KUKA KRL program: di_seitlichFUENFZEHN_unkomp.src, di_seitlichFUENFZEHN_unkomp.dat

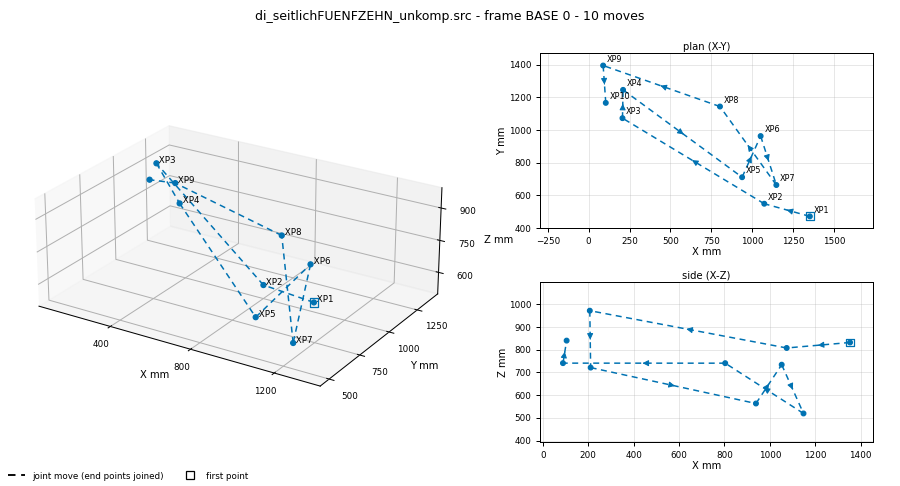
[picture p0: tool path of di_seitlichFUENFZEHN_unkomp.src in frame BASE 0, 10 of 12 moves have a stored position in this frame; points joined in program order, loops and branches not executed]
--- di_seitlichFUENFZEHN_unkomp.src ---
&ACCESS RV
&REL 1
&PARAM EDITMASK = *
&PARAM TEMPLATE = C:\KRC\Roboter\Template\vorgabe
DEF di_s_FZ_unkomp( )
;FOLD INI;%{PE}
  ;FOLD BASISTECH INI
    GLOBAL INTERRUPT DECL 3 WHEN $STOPMESS==TRUE DO IR_STOPM ( )
    INTERRUPT ON 3
    BAS (#INITMOV,0 )
  ;ENDFOLD (BASISTECH INI)
  ;FOLD USER INI
    ;Make your modifications here

  ;ENDFOLD (USER INI)
;ENDFOLD (INI)

;FOLD PTP HOME Vel=10 % DEFAULT;%{PE}%R 8.3.40,%MKUKATPBASIS,%CMOVE,%VPTP,%P 1:PTP, 2:HOME, 3:, 5:10, 7:DEFAULT
$BWDSTART=FALSE
PDAT_ACT=PDEFAULT
FDAT_ACT=FHOME
BAS(#PTP_PARAMS,10)
$H_POS=XHOME
PTP XHOME
;ENDFOLD

WAIT FOR IS_KEY_PRESSED(12)

;FOLD PTP P1 Vel=30 % PDAT1 Tool[11]:jan_ba Base[0];%{PE}%R 8.3.40,%MKUKATPBASIS,%CMOVE,%VPTP,%P 1:PTP, 2:P1, 3:, 5:30, 7:PDAT1
$BWDSTART=FALSE
PDAT_ACT=PPDAT1
FDAT_ACT=FP1
BAS(#PTP_PARAMS,30)
PTP XP1
;ENDFOLD

WAIT FOR IS_KEY_PRESSED(12)

;FOLD PTP P2 Vel=30 % PDAT2 Tool[11]:jan_ba Base[0];%{PE}%R 8.3.40,%MKUKATPBASIS,%CMOVE,%VPTP,%P 1:PTP, 2:P2, 3:, 5:30, 7:PDAT2
$BWDSTART=FALSE
PDAT_ACT=PPDAT2
FDAT_ACT=FP2
BAS(#PTP_PARAMS,30)
PTP XP2
;ENDFOLD

WAIT FOR IS_KEY_PRESSED(12)

;FOLD PTP P3 Vel=30 % PDAT3 Tool[11]:jan_ba Base[0];%{PE}%R 8.3.40,%MKUKATPBASIS,%CMOVE,%VPTP,%P 1:PTP, 2:P3, 3:, 5:30, 7:PDAT3
$BWDSTART=FALSE
PDAT_ACT=PPDAT3
FDAT_ACT=FP3
BAS(#PTP_PARAMS,30)
PTP XP3
;ENDFOLD

WAIT FOR IS_KEY_PRESSED(12)

;FOLD PTP P4 Vel=30 % PDAT4 Tool[11]:jan_ba Base[0];%{PE}%R 8.3.40,%MKUKATPBASIS,%CMOVE,%VPTP,%P 1:PTP, 2:P4, 3:, 5:30, 7:PDAT4
$BWDSTART=FALSE
PDAT_ACT=PPDAT4
FDAT_ACT=FP4
BAS(#PTP_PARAMS,30)
PTP XP4
;ENDFOLD

WAIT FOR IS_KEY_PRESSED(12)

;FOLD PTP P5 Vel=30 % PDAT5 Tool[11]:jan_ba Base[0];%{PE}%R 8.3.40,%MKUKATPBASIS,%CMOVE,%VPTP,%P 1:PTP, 2:P5, 3:, 5:30, 7:PDAT5
$BWDSTART=FALSE
PDAT_ACT=PPDAT5
FDAT_ACT=FP5
BAS(#PTP_PARAMS,30)
PTP XP5
;ENDFOLD

WAIT FOR IS_KEY_PRESSED(12)


;FOLD PTP P6 Vel=30 % PDAT6 Tool[11]:jan_ba Base[0];%{PE}%R 8.3.40,%MKUKATPBASIS,%CMOVE,%VPTP,%P 1:PTP, 2:P6, 3:, 5:30, 7:PDAT6
$BWDSTART=FALSE
PDAT_ACT=PPDAT6
FDAT_ACT=FP6
BAS(#PTP_PARAMS,30)
PTP XP6
;ENDFOLD
WAIT FOR IS_KEY_PRESSED(12)

;FOLD PTP P7 Vel=30 % PDAT7 Tool[11]:jan_ba Base[0];%{PE}%R 8.3.40,%MKUKATPBASIS,%CMOVE,%VPTP,%P 1:PTP, 2:P7, 3:, 5:30, 7:PDAT7
$BWDSTART=FALSE
PDAT_ACT=PPDAT7
FDAT_ACT=FP7
BAS(#PTP_PARAMS,30)
PTP XP7
;ENDFOLD

WAIT FOR IS_KEY_PRESSED(12)

;FOLD PTP P8 Vel=30 % PDAT8 Tool[11]:jan_ba Base[0];%{PE}%R 8.3.40,%MKUKATPBASIS,%CMOVE,%VPTP,%P 1:PTP, 2:P8, 3:, 5:30, 7:PDAT8
$BWDSTART=FALSE
PDAT_ACT=PPDAT8
FDAT_ACT=FP8
BAS(#PTP_PARAMS,30)
PTP XP8
;ENDFOLD

WAIT FOR IS_KEY_PRESSED(12)

;FOLD PTP P9 Vel=30 % PDAT9 Tool[11]:jan_ba Base[0];%{PE}%R 8.3.40,%MKUKATPBASIS,%CMOVE,%VPTP,%P 1:PTP, 2:P9, 3:, 5:30, 7:PDAT9
$BWDSTART=FALSE
PDAT_ACT=PPDAT9
FDAT_ACT=FP9
BAS(#PTP_PARAMS,30)
PTP XP9
;ENDFOLD

WAIT FOR IS_KEY_PRESSED(12)

;FOLD PTP P10 Vel=30 % PDAT10 Tool[11]:jan_ba Base[0];%{PE}%R 8.3.40,%MKUKATPBASIS,%CMOVE,%VPTP,%P 1:PTP, 2:P10, 3:, 5:30, 7:PDAT10
$BWDSTART=FALSE
PDAT_ACT=PPDAT10
FDAT_ACT=FP10
BAS(#PTP_PARAMS,30)
PTP XP10
;ENDFOLD

WAIT FOR IS_KEY_PRESSED(12)

;FOLD PTP HOME Vel=10 % DEFAULT;%{PE}%R 8.3.40,%MKUKATPBASIS,%CMOVE,%VPTP,%P 1:PTP, 2:HOME, 3:, 5:10, 7:DEFAULT
$BWDSTART=FALSE
PDAT_ACT=PDEFAULT
FDAT_ACT=FHOME
BAS(#PTP_PARAMS,10)
$H_POS=XHOME
PTP XHOME
;ENDFOLD

END

--- di_seitlichFUENFZEHN_unkomp.dat ---
&ACCESS RV
&REL 1
&PARAM EDITMASK = *
&PARAM TEMPLATE = C:\KRC\Roboter\Template\vorgabe
DEFDAT  di_s_FZ_unkomp
;FOLD EXTERNAL DECLARATIONS;%{PE}%MKUKATPBASIS,%CEXT,%VCOMMON,%P
;FOLD BASISTECH EXT;%{PE}%MKUKATPBASIS,%CEXT,%VEXT,%P
EXT  BAS (BAS_COMMAND  :IN,REAL  :IN )
DECL INT SUCCESS
;ENDFOLD (BASISTECH EXT)
;FOLD USER EXT;%{E}%MKUKATPUSER,%CEXT,%VEXT,%P
;Make your modifications here

;ENDFOLD (USER EXT)
;ENDFOLD (EXTERNAL DECLARATIONS)
DECL BASIS_SUGG_T LAST_BASIS={POINT1[] "P10                     ",POINT2[] "P10                     ",CP_PARAMS[] "CPDAT0                  ",PTP_PARAMS[] "PDAT10                  ",CONT[] "                        ",CP_VEL[] "2.0                     ",PTP_VEL[] "30                      ",SYNC_PARAMS[] "SYNCDAT                 ",SPL_NAME[] "S0                      ",A_PARAMS[] "ADAT0                   "}
DECL E6POS XP1={X 1353.26367,Y 472.287628,Z 831.916565,A -169.097366,B 77.3817520,C 171.184265,S 22,T 51,E1 0.00522593,E2 20159.9980,E3 0.0,E4 0.0,E5 0.0,E6 0.0}
DECL FDAT FP1={TOOL_NO 11,BASE_NO 0,IPO_FRAME #BASE,POINT2[] " ",TQ_STATE FALSE}
DECL PDAT PPDAT1={VEL 100.000,ACC 50.0000,APO_DIST 100.000,APO_MODE #CDIS,GEAR_JERK 50.0000,EXAX_IGN 0}
DECL E6POS XP2={X 1074.25488,Y 549.450,Z 807.697449,A -99.9409561,B 76.8414764,C -152.987686,S 22,T 51,E1 0.00522593,E2 20159.9980,E3 0.0,E4 0.0,E5 0.0,E6 0.0}
DECL FDAT FP2={TOOL_NO 11,BASE_NO 0,IPO_FRAME #BASE,POINT2[] " ",TQ_STATE FALSE}
DECL PDAT PPDAT2={VEL 100.000,ACC 50.0000,APO_DIST 100.000,APO_MODE #CDIS,GEAR_JERK 50.0000,EXAX_IGN 0}
DECL E6POS XP3={X 206.771683,Y 1073.02307,Z 971.965,A -10.1191072,B 44.6533699,C -91.3017120,S 22,T 19,E1 0.00522593,E2 20159.9980,E3 0.0,E4 0.0,E5 0.0,E6 0.0}
DECL FDAT FP3={TOOL_NO 11,BASE_NO 0,IPO_FRAME #BASE,POINT2[] " ",TQ_STATE FALSE}
DECL PDAT PPDAT3={VEL 100.000,ACC 50.0000,APO_DIST 100.000,APO_MODE #CDIS,GEAR_JERK 50.0000,EXAX_IGN 0}
DECL E6POS XP4={X 210.482193,Y 1246.13611,Z 721.276184,A -6.27344370,B 12.8721447,C -131.382736,S 22,T 19,E1 0.00522593,E2 20159.9980,E3 0.0,E4 0.0,E5 0.0,E6 0.0}
DECL FDAT FP4={TOOL_NO 11,BASE_NO 0,IPO_FRAME #BASE,POINT2[] " ",TQ_STATE FALSE}
DECL PDAT PPDAT4={VEL 100.000,ACC 50.0000,APO_DIST 100.000,APO_MODE #CDIS,GEAR_JERK 50.0000,EXAX_IGN 0}
DECL E6POS XP5={X 938.787537,Y 711.655090,Z 563.083679,A -147.139725,B 70.3353806,C 156.872284,S 22,T 51,E1 0.00522593,E2 20159.9980,E3 0.0,E4 0.0,E5 0.0,E6 0.0}
DECL FDAT FP5={TOOL_NO 11,BASE_NO 0,IPO_FRAME #BASE,POINT2[] " ",TQ_STATE FALSE}
DECL PDAT PPDAT5={VEL 100.000,ACC 50.0000,APO_DIST 100.000,APO_MODE #CDIS,GEAR_JERK 50.0000,EXAX_IGN 0}
DECL E6POS XP6={X 1052.16724,Y 963.509094,Z 734.038635,A 29.0097256,B 71.8549652,C -55.5883713,S 22,T 19,E1 0.00522593,E2 20159.9980,E3 0.0,E4 0.0,E5 0.0,E6 0.0}
DECL FDAT FP6={TOOL_NO 11,BASE_NO 0,IPO_FRAME #BASE,POINT2[] " ",TQ_STATE FALSE}
DECL PDAT PPDAT6={VEL 100.000,ACC 50.0000,APO_DIST 100.000,APO_MODE #CDIS,GEAR_JERK 50.0000,EXAX_IGN 0}
DECL E6POS XP7={X 1148.25061,Y 664.009888,Z 519.207031,A -52.2922440,B 62.4936752,C -126.839088,S 22,T 19,E1 0.00522593,E2 20159.9980,E3 0.0,E4 0.0,E5 0.0,E6 0.0}
DECL FDAT FP7={TOOL_NO 11,BASE_NO 0,IPO_FRAME #BASE,POINT2[] " ",TQ_STATE FALSE}
DECL PDAT PPDAT7={VEL 100.000,ACC 50.0000,APO_DIST 100.000,APO_MODE #CDIS,GEAR_JERK 50.0000,EXAX_IGN 0}
DECL E6POS XP8={X 803.311890,Y 1144.23877,Z 740.702759,A -103.009811,B 70.2966156,C -165.131500,S 22,T 19,E1 0.00522593,E2 20159.9980,E3 0.0,E4 0.0,E5 0.0,E6 0.0}
DECL FDAT FP8={TOOL_NO 11,BASE_NO 0,IPO_FRAME #BASE,POINT2[] " ",TQ_STATE FALSE}
DECL PDAT PPDAT8={VEL 100.000,ACC 50.0000,APO_DIST 100.000,APO_MODE #CDIS,GEAR_JERK 50.0000,EXAX_IGN 0}
DECL E6POS XP9={X 88.5504150,Y 1395.10291,Z 740.855591,A -71.5543289,B 70.3010178,C -165.114258,S 22,T 19,E1 0.00522593,E2 20159.9980,E3 0.0,E4 0.0,E5 0.0,E6 0.0}
DECL FDAT FP9={TOOL_NO 11,BASE_NO 0,IPO_FRAME #BASE,POINT2[] " ",TQ_STATE FALSE}
DECL PDAT PPDAT9={VEL 100.000,ACC 50.0000,APO_DIST 100.000,APO_MODE #CDIS,GEAR_JERK 50.0000,EXAX_IGN 0}
DECL E6POS XP10={X 104.654068,Y 1166.67981,Z 840.163208,A -154.227066,B 84.4587555,C 124.997437,S 22,T 59,E1 0.00522593,E2 20159.9980,E3 0.0,E4 0.0,E5 0.0,E6 0.0}
DECL FDAT FP10={TOOL_NO 11,BASE_NO 0,IPO_FRAME #BASE,POINT2[] " ",TQ_STATE FALSE}
DECL PDAT PPDAT10={VEL 100.000,ACC 50.0000,APO_DIST 100.000,APO_MODE #CDIS,GEAR_JERK 50.0000,EXAX_IGN 0}
ENDDAT
